SYSTEM TANK_VIEWL (* Level Control System View+HMI *)
  (* Standard: 61499-1; Classification: Simulation; ApplicationDomain: Process Control *)
  (* Version 0.1, 2004-09-02, JHC, Rockwell Automation, Separated TANK, VALVE, PUMP resources. *)
  (* Version 0.0, 2004-08-20, JHC, Rockwell Automation, Adapted from DRILL_VIEWL *)
  DEVICE HMI : FRAME_DEVICE(BOUNDS := [100,100,150,120], GRID := [3,1])
    RESOURCE VALVE : PANEL_RESOURCE
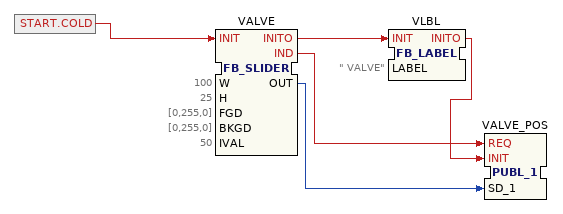
      FBS
        VALVE_POS : PUBL_1;
        VALVE : FB_SLIDER(W := 100, H := 25, FGD := [0,255,0], BKGD := [0,255,0], IVAL := 50);
        VLBL : FB_LABEL(LABEL := " VALVE");
      END_FBS
      EVENT_CONNECTIONS
        START.COLD TO VALVE.INIT;
        VALVE.INITO TO VLBL.INIT;
        VALVE.IND TO VALVE_POS.REQ;
        VLBL.INITO TO VALVE_POS.INIT;
      END_CONNECTIONS
      DATA_CONNECTIONS
        VALVE.OUT TO VALVE_POS.SD_1;
      END_CONNECTIONS
    END_RESOURCE
    RESOURCE TANK : PANEL_RESOURCE
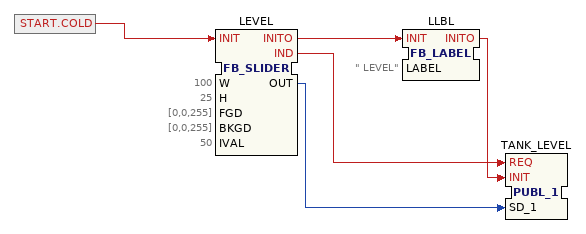
      FBS
        TANK_LEVEL : PUBL_1;
        LEVEL : FB_SLIDER(W := 100, H := 25, FGD := [0,0,255], BKGD := [0,0,255], IVAL := 50);
        LLBL : FB_LABEL(LABEL := " LEVEL");
      END_FBS
      EVENT_CONNECTIONS
        LEVEL.INITO TO LLBL.INIT;
        LEVEL.IND TO TANK_LEVEL.REQ;
        START.COLD TO LEVEL.INIT;
        LLBL.INITO TO TANK_LEVEL.INIT;
      END_CONNECTIONS
      DATA_CONNECTIONS
        LEVEL.OUT TO TANK_LEVEL.SD_1;
      END_CONNECTIONS
    END_RESOURCE
    RESOURCE PUMP : PANEL_RESOURCE
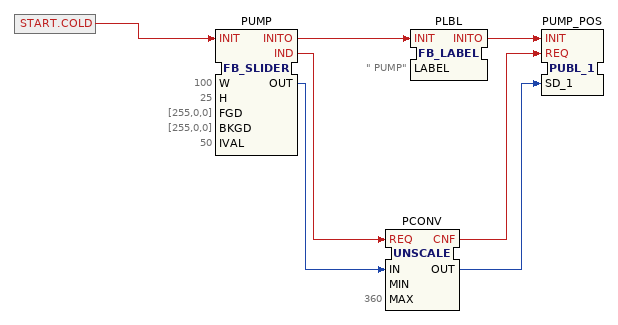
      FBS
        PUMP_POS : PUBL_1;
        PUMP : FB_SLIDER(W := 100, H := 25, FGD := [255,0,0], BKGD := [255,0,0], IVAL := 50);
        PLBL : FB_LABEL(LABEL := " PUMP");
        PCONV : UNSCALE(MAX := 360);
      END_FBS
      EVENT_CONNECTIONS
        PUMP.INITO TO PLBL.INIT;
        PLBL.INITO TO PUMP_POS.INIT;
        PUMP.IND TO PCONV.REQ;
        PCONV.CNF TO PUMP_POS.REQ;
        START.COLD TO PUMP.INIT;
      END_CONNECTIONS
      DATA_CONNECTIONS
        PUMP.OUT TO PCONV.IN;
        PCONV.OUT TO PUMP_POS.SD_1;
      END_CONNECTIONS
    END_RESOURCE
  END_DEVICE
  DEVICE VIEW : FRAME_DEVICE(BOUNDS := [250,100,175,250])
    RESOURCE VALVE : VIEW_PANEL(DIA := 50, SIZE := [1,3])
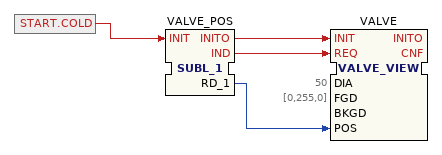
      FBS
        VALVE_POS : SUBL_1;
        VALVE : VALVE_VIEW(DIA := 50, FGD := [0,255,0]);
      END_FBS
      EVENT_CONNECTIONS
        START.COLD TO VALVE_POS.INIT;
        VALVE_POS.INITO TO VALVE.INIT;
        VALVE_POS.IND TO VALVE.REQ;
      END_CONNECTIONS
      DATA_CONNECTIONS
        VALVE_POS.RD_1 TO VALVE.POS;
      END_CONNECTIONS
    END_RESOURCE
    RESOURCE TANK : VIEW_PANEL(SIZE := [1,2], DIA := 75)
      FBS
        TANK : MECH_VIEW(STYLE := VSTYLE#CYLINDER, LEN := 2, DIR := 3, BKGD := [255,255,255], WKPC := [0,0,255]);
        TANK_LEVEL : SUBL_1;
      END_FBS
      EVENT_CONNECTIONS
        TANK_LEVEL.INITO TO TANK.INIT;
        TANK_LEVEL.IND TO TANK.REQ;
        START.COLD TO TANK_LEVEL.INIT;
      END_CONNECTIONS
      DATA_CONNECTIONS
        TANK_LEVEL.RD_1 TO TANK.POS;
      END_CONNECTIONS
    END_RESOURCE
    RESOURCE PUMP : VIEW_PANEL(DIA := 50, SIZE := [4,1])
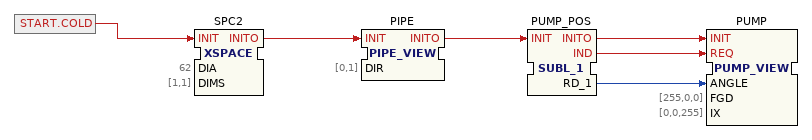
      FBS
        PUMP_POS : SUBL_1;
        SPC2 : XSPACE(DIA := 62, DIMS := [1,1]);
        PIPE : PIPE_VIEW(DIR := [0,1]);
        PUMP : PUMP_VIEW(FGD := [255,0,0], IX := [0,0,255]);
      END_FBS
      EVENT_CONNECTIONS
        SPC2.INITO TO PIPE.INIT;
        START.COLD TO SPC2.INIT;
        PIPE.INITO TO PUMP_POS.INIT;
        PUMP_POS.INITO TO PUMP.INIT;
        PUMP_POS.IND TO PUMP.REQ;
      END_CONNECTIONS
      DATA_CONNECTIONS
        PUMP_POS.RD_1 TO PUMP.ANGLE;
      END_CONNECTIONS
    END_RESOURCE
  END_DEVICE
END_SYSTEM
